INTERFACE I_Mover

METHOD CycleUpdate : BOOL
VAR_INPUT

END_VAR
END_METHOD

PROPERTY distToEndOfTrack : LREAL
GET
END_GET
END_PROPERTY

METHOD Init : BOOL
VAR_INPUT
	XtsMover:  I_XtsXlMover1;
	XtsProcessingUnit :  I_XtsProcessingUnit1;
END_VAR
END_METHOD

METHOD JoinNearestTrack : BOOL


VAR

END_VAR
END_METHOD

METHOD LeaveSystemAt : BOOL
VAR_INPUT
	ConnectionOut: REFERENCE TO MC_PlanarTrackConnectionOut;	
END_VAR
END_METHOD

METHOD MoveOnTrack : BOOL
VAR_INPUT
	track: REFERENCE TO MC_PlanarTrack;	
	targetPos: LREAL;	
	gap: LREAL;

END_VAR
END_METHOD

PROPERTY MoverStopped : BOOL
GET
END_GET
SET
END_SET
END_PROPERTY

PROPERTY P_Dynamics : REFERENCE TO DynamicConstraint_PathXY;
GET
END_GET
END_PROPERTY

PROPERTY P_MoveOnTrackOptions : REFERENCE TO ST_MoveOnTrackOptions;
GET
END_GET
END_PROPERTY

PROPERTY P_MoverOTCID : OTCID
GET
END_GET
END_PROPERTY

PROPERTY P_PlanarFeedback : REFERENCE TO MC_PlanarFeedback
GET
END_GET
END_PROPERTY

PROPERTY P_PlanarMover :   REFERENCE TO  MC_PlanarMover
GET
END_GET
END_PROPERTY

PROPERTY P_SyncFeedback : REFERENCE TO MC_PlanarFeedbackGearInPosOnTrackWithMasterMover
GET
END_GET
END_PROPERTY

PROPERTY P_TargetTrack : UDINT
GET
END_GET
SET
END_SET
END_PROPERTY

PROPERTY Rework : BOOL
GET
END_GET
SET
END_SET
END_PROPERTY

METHOD SyncToOtherMover : Bool
VAR_INPUT
	masterSyncPos : LREAL; // Position on the master track
	followerSyncPos : LREAL; // position on the follower track
	PlanarMoverToFollow: REFERENCE TO Tc3_Mc3PlanarMotion.MC_PlanarMover;
	masterTrack : REFERENCE TO Tc3_Mc3PlanarMotion.MC_PlanarTrack; 
	followerTrack : REFERENCE TO Tc3_Mc3PlanarMotion.MC_PlanarTrack; 
	velo : LREAL; 
END_VAR
END_METHOD

METHOD  UpdateXtsTrack
VAR_INPUT
END_VAR
VAR

END_VAR
END_METHOD

PROPERTY XlProcessingUnit : I_XtsProcessingUnit1
GET
END_GET
END_PROPERTY

PROPERTY XtsComFeed : REFERENCE TO  XtsCommandFeedback
GET
END_GET
END_PROPERTY

PROPERTY XtsXlMover :  I_XtsXlMover1
GET
END_GET
END_PROPERTY

END_INTERFACE

(* stored: Version 1.1.0.1, ProductVersion 3.1.4026.8
   Itf I_Mover: Id {8f7a23e9-9aaf-41cd-ab60-e1f3e7434be6}
   Method CycleUpdate: Id {16b91d1c-6612-4b15-8ad2-636991d1ec4b}
   Property distToEndOfTrack: Id {fb9918b4-0722-48f8-b168-52aeaaa03f02}
   Get Get: Id {433eaf7b-763b-4281-b0de-2d687b311edb}
   Method Init: Id {7d28287b-661a-454a-bbbf-866a25751a67}
   Method JoinNearestTrack: Id {fcd27990-deab-4421-b7b8-1b953f6ea6ad}
   Method LeaveSystemAt: Id {6f2a2cbe-473d-4242-8909-5b4e3f2617b3}
   Method MoveOnTrack: Id {c13e8780-a810-4cef-9f66-33ce7886d601}
   Property MoverStopped: Id {cf4e5790-f4c7-4a34-a6b7-f827bd1b58ea}
   Get Get: Id {73e4d349-958f-49aa-8819-82dc54fcaf7e}
   Set Set: Id {2984a813-2861-404e-afcd-6fe40b3f298b}
   Property P_Dynamics: Id {49f87732-ac80-4370-864b-d299b8982fb4}
   Get Get: Id {903e88f0-856c-40e6-82b1-4d7fd487c3a1}
   Property P_MoveOnTrackOptions: Id {58176a06-420f-43c2-97e9-0a0866e730ae}
   Get Get: Id {6b0efbc1-c933-4562-829f-485e4cd01185}
   Property P_MoverOTCID: Id {7aee9de3-dd1b-4cf1-919f-0b06c2a67455}
   Get Get: Id {72dd4685-dec2-4ec6-a1f9-7c5baddcbdbd}
   Property P_PlanarFeedback: Id {a9bbed57-3b9f-4517-b2ea-da5c58571634}
   Get Get: Id {1f34cbf7-27f6-4e1e-bf7e-6065ca290696}
   Property P_PlanarMover: Id {251d31a4-2c02-4df5-94c5-20fa73edfdf1}
   Get Get: Id {a86b8714-3613-43d4-90ac-0b1a90218c8d}
   Property P_SyncFeedback: Id {44e12130-9d7b-42f1-8fbe-83c3e8bf9e21}
   Get Get: Id {c1e62b68-c344-428b-816f-4dc4e05c9105}
   Property P_TargetTrack: Id {5f388733-1fb3-404b-a5dd-52830cf45c04}
   Get Get: Id {809a5c07-54f0-4fe3-aefb-7e900f64f163}
   Set Set: Id {3d5b627b-7e6a-4502-b473-8d3ae7ff12bc}
   Property Rework: Id {3fe0cb1d-a009-4172-baa6-bc56de96dde9}
   Get Get: Id {ae6b01cc-d3e1-4ca8-a0ef-10aa8b8616ec}
   Set Set: Id {c35d6475-d359-4b71-b6dc-7aa7369c8609}
   Method SyncToOtherMover: Id {53951dae-e642-4c0f-afd2-22812dd067a9}
   Method UpdateXtsTrack: Id {5fee0b6d-2168-4518-a132-30a77a73fb31}
   Property XlProcessingUnit: Id {dd82962b-2ee3-41c8-88b9-f5400df6df47}
   Get Get: Id {5f7bca70-5352-4656-adad-72b4bfd0f749}
   Property XtsComFeed: Id {6c7b5599-6bad-4746-b79f-cc3b776015d0}
   Get Get: Id {f07767b0-f530-48d2-a8fa-343aaf046073}
   Property XtsXlMover: Id {52294691-411d-487f-bcfb-f7b79c0a9bc7}
   Get Get: Id {830996b0-f731-49d4-af8d-f3122d44d6e6} *)
